// TwinCAT 3 PLC project PLCStudent
// ProgramVersion: 3.1.4026.20
// libraries:
//   Tc2_Standard, * (Beckhoff Automation GmbH)
//   Tc2_System, * (Beckhoff Automation GmbH)
//   Tc2_Utilities, * (Beckhoff Automation GmbH)
//   Tc3_IotBase, * (Beckhoff Automation GmbH)
//   Tc3_JsonXml, * (Beckhoff Automation GmbH)
//   Tc3_Module, * (Beckhoff Automation GmbH)
//   VisuSymbols, 4.5.0.0 (System)
// project tree:
//   / GlobalTextList.TcGTLO, PlcTask.TcTTO, Visualization Manager.TcVMO (not stored)
//   GVLs/ GVL.TcGVL
//   POUs/ FB_HTTP_Get.TcPOU, FB_HTTP_GetSafety.TcPOU, FB_HTTP_Post.TcPOU, FB_OrderAGV.TcPOU, FB_ParseJsonResponse.TcPOU, MAIN.TcPOU, OrderRobot.TcPOU, Process.TcPOU
//   VISUs/ Visualization.TcVIS
// (motion and I/O tree: see PLC project plcsim)
// real-time tasks:
//   TASK PlcTask: cycle T#20ms, priority 20, ADS port 350
// variable links:
//   PLCSim/PLCSim Instance <-> PLCStudent/PLCStudent Instance
//     PlcTask Inputs/GVL.iiGotoPos <-> PlcTask Outputs/GVL.qiGotoPos
//     PlcTask Inputs/GVL.ixPLCStrobe <-> PlcTask Outputs/GVL.qxPLCStrobe
//     PlcTask Outputs/GVL.qiAtPos <-> PlcTask Inputs/GVL.iiAtPos
//     PlcTask Outputs/GVL.qxAGVStrobe <-> PlcTask Inputs/GVL.ixAGVStrobe

CONFIGURATION PLCStudent
    RESOURCE PLC ON TwinCAT3
        TASK PlcTask(INTERVAL := T#20ms, PRIORITY := 20);
        PROGRAM MAIN WITH PlcTask : MAIN;
    END_RESOURCE
END_CONFIGURATION

// ---- GVLs/GVL.TcGVL
{attribute 'qualified_only'}
VAR_GLOBAL
//Input to PLC from process
	ixAGVStrobe		AT %I*:	BOOL;	(* AGV strobe signal *)
	iiAtPos			AT %I*:	INT;	(* Actual position of AGV *)
	
//Output from PLC to process
	qxPLCStrobe		AT %Q*:	BOOL;	(* PLC strobe signal *)
	qiGotoPos		AT %Q*:	INT;	(* Target position for AGV *)
// ADD THESE for R1 route control
    xStart         : BOOL := FALSE;
    iOrder         : INT  := 0;
    xStop          : BOOL := FALSE;
	OrderRobot_0   : OrderRobot;
// R2 data transmission
    sLocation      : STRING := '';
    iBattery       : INT    := 75;
    xSendNow       : BOOL   := FALSE;
END_VAR

// ---- POUs/MAIN.TcPOU
PROGRAM MAIN
VAR
    (* R1: Route state machine *)
    iRouteState     : INT := 0;
    iBattery        : INT := 100;

    (* R2: HTTP POST *)
    fbHttpClientPost : FB_IotHttpClient := (
        sHostName          := '127.0.0.1',
        nHostPort          := 5000,
        bKeepAlive         := TRUE,
        tConnectionTimeout := T#10S
    );
    fbPost      : FB_HTTP_Post;
    bSendPost   : BOOL := FALSE;
    sLocation   : STRING;
   fbFormat : FB_FormatString;
    (* R2: Timestamp *)
    fbTime      : FB_LocalSystemTime := (bEnable := TRUE, dwCycle := 1);
    sTimeStamp  : STRING;

    (* R4: Safety check *)
    fbHttpClientGet : FB_IotHttpClient := (
        sHostName          := '127.0.0.1',
        nHostPort          := 5000,
        bKeepAlive         := TRUE,
        tConnectionTimeout := T#10S
    );
    fbSafetyCheck   : FB_HTTP_GetSafety;
    bSendSafety     : BOOL := FALSE;
    safetyPollTimer : TON;
    sNextLocation   : STRING;
END_VAR

(* R2: 每个周期构建时间戳 *)
fbTime(bEnable := TRUE, dwCycle := 1);
fbFormat(
    sFormat := '%d-%02d-%02d %02d:%02d:%02d', 
    arg1 := F_WORD(fbTime.systemTime.wYear),
    arg2 := F_WORD(fbTime.systemTime.wMonth),
    arg3 := F_WORD(fbTime.systemTime.wDay),
    arg4 := F_WORD(fbTime.systemTime.wHour),
    arg5 := F_WORD(fbTime.systemTime.wMinute),
    arg6 := F_WORD(fbTime.systemTime.wSecond),
    sOut => sTimeStamp
);
CASE iRouteState OF

    (* ────────────────────────────────── *)
    (* 启动阶段                            *)
    (* ────────────────────────────────── *)
    0: (* 启动 — 首先返回原点(Home) *)
        GVL.iOrder  := 1;
        GVL.xStart  := TRUE;
        iRouteState := 10;

    10: (* 等待 AGV 到达原点 *)
        GVL.xStart := FALSE;
        IF GVL.OrderRobot_0.iPhase = 0 THEN
            iRouteState := 12;
        END_IF

    (* ────────────────────────────────── *)
    (* 位置 A                             *)
    (* ────────────────────────────────── *)
    11: (* 前往位置 A *)
        GVL.iOrder  := 2;
        GVL.xStart  := TRUE;
        iRouteState := 20;

    (* ────────────────────────────────── *)
    (* 安全检查 A                         *)
    (* ────────────────────────────────── *)
    12: (* 设置位置，复位发送信号 *)
        sNextLocation := 'A';
        bSendSafety   := FALSE;
        iRouteState   := 13;

    13: (* 发送持续一个周期的脉冲信号 *)
        bSendSafety := TRUE;
        iRouteState := 14;

    14: (* 等待位置 A 的安全检查结果 *)
        bSendSafety := FALSE;
        IF fbSafetyCheck.bDone THEN 
            IF fbSafetyCheck.bIsSafe THEN
                safetyPollTimer(IN := FALSE);
                iRouteState := 11;      (* 安全 → 前往位置 A *)
            ELSE
                (* 不安全 → 等待 2 秒后重试 *)
                safetyPollTimer(IN := TRUE, PT := T#2S);
                IF safetyPollTimer.Q THEN
                    safetyPollTimer(IN := FALSE);
                    iRouteState := 12;  (* 重试 *)
                END_IF
            END_IF
        ELSE
            (* 未收到完成信号 (bDone) → 5 秒后超时 *)
            safetyPollTimer(IN := TRUE, PT := T#5S);
            IF safetyPollTimer.Q THEN
                safetyPollTimer(IN := FALSE);
                iRouteState := 12;      (* 从头重试 *)
            END_IF
        END_IF



    20: (* AGV 已到达位置 A *)
        GVL.xStart := FALSE;
        IF GVL.OrderRobot_0.iPhase = 0 THEN
            sLocation   := 'A';
            iBattery    := iBattery - 5;
            bSendPost   := TRUE;
            iRouteState := 25;
        END_IF

    25: (* 等待位置 A 的 POST 数据上报完成 *)
        bSendPost := FALSE;
        IF NOT fbPost.bBusy THEN
            iRouteState := 26;
        END_IF

    (* ────────────────────────────────── *)
    (* 安全检查 B                         *)
    (* ────────────────────────────────── *)
    26: (* 设置位置，复位发送信号 *)
        sNextLocation := 'B';
        bSendSafety   := FALSE;
        iRouteState   := 27;

    27: (* 发送持续一个周期的脉冲信号 *)
        bSendSafety := TRUE;
        iRouteState := 28;

    28: (* 等待位置 B 的安全检查结果 *)
        bSendSafety := FALSE;
        IF fbSafetyCheck.bDone THEN
            IF fbSafetyCheck.bIsSafe THEN
                safetyPollTimer(IN := FALSE);
                iRouteState := 21;      (* 安全 → 前往位置 B *)
            ELSE
                (* 不安全 → 等待 2 秒后重试 *)
                safetyPollTimer(IN := TRUE, PT := T#2S);
                IF safetyPollTimer.Q THEN
                    safetyPollTimer(IN := FALSE);
                    iRouteState := 26;  (* 重试 *)
                END_IF
            END_IF
        ELSE
            (* 未收到完成信号 (bDone) → 5 秒后超时 *)
            safetyPollTimer(IN := TRUE, PT := T#5S);
            IF safetyPollTimer.Q THEN
                safetyPollTimer(IN := FALSE);
                iRouteState := 26;      (* 从头重试 *)
            END_IF
        END_IF

    (* ────────────────────────────────── *)
    (* 位置 B                             *)
    (* ────────────────────────────────── *)
    21: (* 前往位置 B *)
        GVL.iOrder  := 3;
        GVL.xStart  := TRUE;
        iRouteState := 30;

    30: (* AGV 已到达位置 B *)
        GVL.xStart := FALSE;
        IF GVL.OrderRobot_0.iPhase = 0 THEN
            sLocation   := 'B';
            iBattery    := iBattery - 5;
            bSendPost   := TRUE;
            iRouteState := 35;
        END_IF

    35: (* 等待位置 B 的 POST 数据上报完成 *)
        bSendPost := FALSE;
        IF NOT fbPost.bBusy THEN
            iRouteState := 36;
        END_IF

    (* ────────────────────────────────── *)
    (* 安全检查 C                         *)
    (* ────────────────────────────────── *)
    36: (* 设置位置，复位发送信号 *)
        sNextLocation := 'C';
        bSendSafety   := FALSE;
        iRouteState   := 37;

    37: (* 发送持续一个周期的脉冲信号 *)
        bSendSafety := TRUE;
        iRouteState := 38;

    38: (* 等待位置 C 的安全检查结果 *)
        bSendSafety := FALSE;
        IF fbSafetyCheck.bDone THEN
            IF fbSafetyCheck.bIsSafe THEN
                safetyPollTimer(IN := FALSE);
                iRouteState := 31;      (* 安全 → 前往位置 C *)
            ELSE
                (* 不安全 → 等待 2 秒后重试 *)
                safetyPollTimer(IN := TRUE, PT := T#2S);
                IF safetyPollTimer.Q THEN
                    safetyPollTimer(IN := FALSE);
                    iRouteState := 36;  (* 重试 *)
                END_IF
            END_IF
        ELSE
            (* 未收到完成信号 (bDone) → 5 秒后超时 *)
            safetyPollTimer(IN := TRUE, PT := T#5S);
            IF safetyPollTimer.Q THEN
                safetyPollTimer(IN := FALSE);
                iRouteState := 36;      (* 从头重试 *)
            END_IF
        END_IF

    (* ────────────────────────────────── *)
    (* 位置 C                             *)
    (* ────────────────────────────────── *)
    31: (* 前往位置 C *)
        GVL.iOrder  := 4;
        GVL.xStart  := TRUE;
        iRouteState := 40;

    40: (* AGV 已到达位置 C *)
        GVL.xStart := FALSE;
        IF GVL.OrderRobot_0.iPhase = 0 THEN
            sLocation   := 'C';
            iBattery    := iBattery - 5;
            bSendPost   := TRUE;
            iRouteState := 45;
        END_IF

    45: (* 等待位置 C 的 POST 数据上报完成 *)
        bSendPost := FALSE;
        IF NOT fbPost.bBusy THEN
            iRouteState := 46;
        END_IF

    (* ────────────────────────────────── *)
    (* 安全检查 D                         *)
    (* ────────────────────────────────── *)
    46: (* 设置位置，复位发送信号 *)
        sNextLocation := 'D';
        bSendSafety   := FALSE;
        iRouteState   := 47;

    47: (* 发送持续一个周期的脉冲信号 *)
        bSendSafety := TRUE;
        iRouteState := 48;

    48: (* 等待位置 D 的安全检查结果 *)
        bSendSafety := FALSE;
        IF fbSafetyCheck.bDone THEN
            IF fbSafetyCheck.bIsSafe THEN
                safetyPollTimer(IN := FALSE);
                iRouteState := 41;      (* 安全 → 前往位置 D *)
            ELSE
                (* 不安全 → 等待 2 秒后重试 *)
                safetyPollTimer(IN := TRUE, PT := T#2S);
                IF safetyPollTimer.Q THEN
                    safetyPollTimer(IN := FALSE);
                    iRouteState := 46;  (* 重试 *)
                END_IF
            END_IF
        ELSE
            (* 未收到完成信号 (bDone) → 5 秒后超时 *)
            safetyPollTimer(IN := TRUE, PT := T#5S);
            IF safetyPollTimer.Q THEN
                safetyPollTimer(IN := FALSE);
                iRouteState := 46;      (* 从头重试 *)
            END_IF
        END_IF

    (* ────────────────────────────────── *)
    (* 位置 D                             *)
    (* ────────────────────────────────── *)
    41: (* 前往位置 D *)
        GVL.iOrder  := 5;
        GVL.xStart  := TRUE;
        iRouteState := 50;

    50: (* AGV 已到达位置 D *)
        GVL.xStart := FALSE;
        IF GVL.OrderRobot_0.iPhase = 0 THEN
            sLocation   := 'D';
            iBattery    := iBattery - 5;
            bSendPost   := TRUE;
            iRouteState := 55;
        END_IF

    55: (* 等待位置 D 的 POST 数据上报完成 *)
        bSendPost := FALSE;
        IF NOT fbPost.bBusy THEN
            iRouteState := 51;
        END_IF

    (* ────────────────────────────────── *)
    (* 返回原点                            *)
    (* ────────────────────────────────── *)
    51: (* 返回原点(Home) *)
        GVL.iOrder  := 1;
        GVL.xStart  := TRUE;
        iRouteState := 60;

    60: (* AGV 已到达原点 — 进行充电 *)
        GVL.xStart := FALSE;
        IF GVL.OrderRobot_0.iPhase = 0 THEN
            sLocation   := 'Home';
            iBattery    := 100;
            bSendPost   := TRUE;
            iRouteState := 65;
        END_IF

    65: (* 等待原点的 POST 数据上报完成 — 再次进入循环 *)
        bSendPost := FALSE;
        IF NOT fbPost.bBusy THEN
            iRouteState := 12;  (* 从位置 A 的安全检查重新开始循环 *)
        END_IF

END_CASE

(* ────────────────────────────────────── *)
(* 始终在每个周期执行                      *)
(* ────────────────────────────────────── *)
fbHttpClientPost.Execute();
fbHttpClientGet.Execute();

fbPost(
    bSend    := bSendPost,
    position := sLocation,
    dateTime := sTimeStamp,
    battery  := iBattery,
    fbClient := fbHttpClientPost
);

fbSafetyCheck(
    bSend     := bSendSafety,
    sLocation := sNextLocation,
    fbClient  := fbHttpClientGet
);

Process();

END_PROGRAM

// ---- POUs/FB_HTTP_Post.TcPOU
FUNCTION_BLOCK FB_HTTP_Post
VAR_INPUT
    bSend           : BOOL;             //Trigger send message
    position        : STRING;           //Location A, B, C, D, Home
    dateTime        : STRING;           //Timestamp
    battery         : INT;              //Battery level
END_VAR
VAR_IN_OUT
    fbClient        : FB_IotHttpClient;
END_VAR
VAR_OUTPUT
    bBusy           : BOOL;
    bError          : BOOL;
    nResCount       : UDINT;
    nOutputStatusCode : UINT;
    sOutputMessage  : STRING(511);
END_VAR
VAR
    fbRequest       : FB_IotHttpRequest;
    fbJson          : FB_JsonDomParser;
    fbPayload       : FB_JsonSaxWriter;
    fbHeader        : FB_IotHttpHeaderFieldMap;
    RisingEdge      : R_TRIG;
    nState          : UDINT;
    bGetContentResult : BOOL;
    sContent        : STRING(511);
    nReqCount       : UDINT;
    nErrCount       : UDINT;
    LoggMessage     : STRING;
	sBattery : STRING;
END_VAR

RisingEdge(CLK:= bSend);
CASE nState OF
0:
    IF RisingEdge.Q THEN
        sContent := DELETE(STR:=sContent, LEN:=511, POS:=1);
        fbPayload.ResetDocument();
        fbPayload.StartObject();
        fbHeader.AddField('Content-Type', 'application/json', FALSE);

        (* Position *)
        fbPayload.AddKey('Position');
        fbPayload.AddString(position);

        (* TimeStamp — no colon! *)
        fbPayload.AddKey('TimeStamp');
        fbPayload.AddString(dateTime);

        (* Battery — NEW *)
        sBattery := INT_TO_STRING(battery);
        fbPayload.AddKey('Battery');
        fbPayload.AddString(sBattery);

        fbPayload.EndObject();
        sContent := fbPayload.GetDocument();

        IF fbRequest.SendRequest(
            sUri         := '/post_data',
            fbClient     := fbClient,
            eRequestType := ETcIotHttpRequestType.HTTP_POST,
            pContent     := ADR(sContent),
            nContentSize := LEN2(ADR(sContent)),
            fbHeader) THEN

            nState   := 1;
            IF nReqCount > 10 THEN
                nReqCount := 0;
            END_IF
            nReqCount := nReqCount + 1;
            bBusy     := TRUE;
            bError    := FALSE;
        END_IF
    END_IF

1:
    IF NOT fbRequest.bBusy THEN
        bError            := TRUE;
        nOutputStatusCode := fbRequest.nStatusCode;

        IF NOT fbRequest.bError THEN
            bGetContentResult := fbRequest.GetContent(
                pContent           := ADR(sContent),
                nContentSize       := SIZEOF(sContent),
                bSetNullTermination := TRUE);

            sOutputMessage := sContent;

            IF fbRequest.nStatusCode >= 200 AND fbRequest.nStatusCode < 300 THEN
                bError    := FALSE;
                nResCount := nResCount + 1;
                bBusy     := FALSE;
            END_IF
        END_IF

        nState := 0;
        IF bError THEN
            nErrCount := nErrCount + 1;
        END_IF
    END_IF
END_CASE

END_FUNCTION_BLOCK

// ---- POUs/FB_HTTP_GetSafety.TcPOU
FUNCTION_BLOCK FB_HTTP_GetSafety
VAR_INPUT
    bSend           : BOOL;
    sLocation       : STRING;    (* Pass 'A', 'B', 'C' or 'D' *)
END_VAR
VAR_IN_OUT
    fbClient        : FB_IotHttpClient;
END_VAR
VAR_OUTPUT
    bBusy           : BOOL;
    bError          : BOOL;
    bDone           : BOOL;
    nOutputStatusCode : UINT;
    bIsSafe         : BOOL;      (* TRUE = safe, FALSE = unsafe *)
END_VAR
VAR
    fbRequest       : FB_IotHttpRequest;
    fbJson          : FB_JsonDomParser;
    nState          : UDINT;
    RisingEdge      : R_TRIG;
    jsonDoc         : SJsonValue;
    jsonVal         : SJsonValue;
    sResultValue    : STRING;
    sFullUri        : STRING;
    LoggMessage     : STRING;
END_VAR

RisingEdge(CLK := bSend);  // 调用上升沿检测功能块，把输入CLK绑定到bSend信号，用于检测从FALSE→TRUE的瞬间

CASE nState OF   // 状态机，根据当前状态nState执行不同逻辑

0:  // 状态0：空闲/准备发送请求状态
    bDone := FALSE;  // 标记当前任务尚未完成（每次进入初始状态都清零完成标志）
    
    IF RisingEdge.Q THEN  // 如果检测到bSend的上升沿（触发一次请求）
        
        (* Only path, not full URL *)  // 注释说明这里只拼接路径，不是完整URL
        sFullUri := CONCAT('/get_safety/', sLocation);  // 拼接请求路径，例如 /get_safety/A1

        IF fbRequest.SendRequest(  // 调用HTTP请求发送函数
            sUri         := sFullUri,  // 请求的URI路径
            fbClient     := fbClient,  // HTTP客户端实例
            eRequestType := ETcIotHttpRequestType.HTTP_GET,  // 请求类型：GET
            0, 0, 0)  // 额外参数（未使用，占位）
        THEN  // 如果请求成功发起（注意：只是“发出去”，不是“收到响应”）
            
            nState := 1;  // 切换到状态1（等待响应）
            bBusy  := TRUE;  // 标记系统正在忙（请求处理中）
            bError := FALSE;  // 清除错误标志
            bDone  := FALSE;  // 再次确认未完成（其实这里有点重复）

            ADSLOGSTR(  // TwinCAT日志输出函数
                msgCtrlMask := ADSLOG_MSGTYPE_HINT,  // 日志类型：提示信息
                msgFmtStr   := 'SafetyCheck: Sending request for location %s',  // 日志格式字符串
                strArg      := sLocation  // 替换%s的参数（位置名）
            );
        END_IF
    END_IF

1:  // 状态1：等待HTTP响应完成
    IF NOT fbRequest.bBusy THEN  // 如果请求已经处理完成（不再忙）
        
        nOutputStatusCode := fbRequest.nStatusCode;  // 保存HTTP返回状态码（例如200、404等）

        IF NOT fbRequest.bError AND  // 如果请求过程中没有错误
           fbRequest.nStatusCode >= 200 AND  // 且HTTP状态码在200以上
           fbRequest.nStatusCode < 300  // 且小于300（表示成功响应）
        THEN
            
            jsonDoc := fbRequest.GetJsonDomContent(fbJson);  // 解析HTTP响应内容为JSON DOM结构

            IF jsonDoc <> 0 THEN  // 如果JSON解析成功（非空指针）
                
                (* server.py returns {"safe": "true"} or {"safe": "false"} *)  // 服务端返回格式说明
                
                jsonVal      := fbJson.FindMember(jsonDoc, 'safe');  // 在JSON中查找字段 "safe"
                sResultValue := fbJson.GetString(jsonVal);  // 获取该字段的字符串值（"true" 或 "false"）

                IF sResultValue = 'true' THEN  // 如果返回值是字符串"true"
                    bIsSafe := TRUE;  // 标记为安全
                ELSE  // 否则（包括"false"或异常情况）
                    bIsSafe := FALSE;  // 标记为不安全
                END_IF

                LoggMessage := sResultValue;  // 保存结果字符串用于日志输出
                
                ADSLOGSTR(  // 输出日志
                    msgCtrlMask := ADSLOG_MSGTYPE_HINT,  // 提示类型日志
                    msgFmtStr   := 'SafetyCheck result: %s',  // 日志格式
                    strArg      := LoggMessage  // 输出实际返回值
                );
            ELSE  // 如果JSON解析失败
                
                bIsSafe := FALSE;  // 默认认为不安全（保守处理）
                bError  := TRUE;  // 标记发生错误
            END_IF
        
        ELSE  // 如果请求失败（HTTP错误或通信错误）
            
            bIsSafe := FALSE;  // 默认不安全
            bError  := TRUE;  // 标记错误
        END_IF

        bDone  := TRUE;  // 标记任务完成（无论成功失败都会置TRUE）
        bBusy  := FALSE;  // 清除忙状态
        nState := 0;  // 回到初始状态，等待下一次触发
    END_IF

END_CASE  // 状态机结束

END_FUNCTION_BLOCK

// ---- POUs/Process.TcPOU
PROGRAM Process
VAR
	OrderRobot_0: OrderRobot;
	xStart: BOOL;
	iOrder: INT;
	xStop: BOOL;
END_VAR

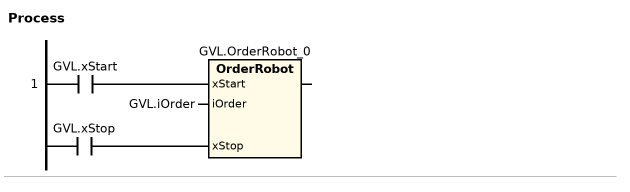
// NETWORK 1
GVL.OrderRobot_0(xStart := GVL.xStart, iOrder := GVL.iOrder, xStop := GVL.xStop); // OrderRobot

END_PROGRAM

// ---- POUs/OrderRobot.TcPOU
FUNCTION_BLOCK OrderRobot
VAR_INPUT
	xStart: BOOL;
	iOrder: INT;
	xStop: BOOL;
END_VAR
VAR_OUTPUT
END_VAR
VAR
	iPhase: INT:=0; //0: Wait signal
END_VAR

CASE iPhase OF
	0: // Wait signal
		IF xStart AND (iOrder<>0) THEN
			iPhase:=1;
		END_IF
	1: // Set Order, here you can add more checking of the numbers are legal or not
		GVL.qiGotoPos:=iOrder;
		iPhase:=2;
	2: // Set strobe
		GVL.qxPLCStrobe:=TRUE;
		iPhase:=3;
	3: // Wait for input strobe
		IF gvl.ixAGVStrobe THEN
			gvl.qiGotoPos:=0;
			gvl.qxPLCStrobe:=FALSE;
			iPhase:=4;
		END_IF
	4: // wait for order finish or stop
		IF xStop THEN
			iPhase:=5;
		ELSIF gvl.iiAtPos<>0 THEN
			iPhase:=6;
		END_IF
	5: // Try to stop
		gvl.qiGotoPos:=6;
		iPhase:=12;
	6: //Wait strobe
		IF gvl.ixAGVStrobe THEN
			iPhase:=7;
		END_IF
	7: // Set strobe
		gvl.qxPLCStrobe:=TRUE;
		iPhase:=8;
	8: // wait for reset
		IF gvl.iiAtPos=0 AND (NOT gvl.ixAGVStrobe) THEN
			gvl.qxPLCStrobe:=FALSE;
			iphase:=0;
		END_IF
	12: // Set strobe
		GVL.qxPLCStrobe:=TRUE;
		iPhase:=13;
	13: // Wait for input strobe
		IF gvl.ixAGVStrobe THEN
			gvl.qiGotoPos:=0;
			gvl.qxPLCStrobe:=FALSE;
			iPhase:=14;
		END_IF
	14: // wait for order finish or stop
		IF gvl.iiAtPos=6 THEN
			iPhase:=16;
		END_IF
	16: //Wait strobe
		IF gvl.ixAGVStrobe THEN
			iPhase:=17;
		END_IF
	17: // Set strobe
		gvl.qxPLCStrobe:=TRUE;
		iPhase:=18;
	18: // wait for reset
		IF gvl.iiAtPos=0 AND (NOT gvl.ixAGVStrobe) THEN
			gvl.qxPLCStrobe:=FALSE;
			iphase:=19;
		END_IF
	19: // Go home
		GVL.qiGotoPos:=1;
		iPhase:=2;
END_CASE

END_FUNCTION_BLOCK

// ---- POUs/FB_HTTP_Get.TcPOU
FUNCTION_BLOCK FB_HTTP_Get
VAR_INPUT
	bSend				: BOOL;
END_VAR
VAR_IN_OUT
	fbClient			: FB_IotHttpClient;
END_VAR	
VAR_OUTPUT
	bBusy				: BOOL;
	bError				: BOOL;
	nOutputStatusCode   : UINT;
	sOutputMessage      : STRING(511);
END_VAR
VAR	
	fbRequest			: FB_IotHttpRequest;
	fbJson				: FB_JsonDomParser;
	jsonMember       : SJsonValue;
	fbHeader: FB_IotHttpHeaderFieldMap;
	nState				: UDINT;
	RisingEdge			: R_TRIG;
	
	bGetContentResult	: BOOL;
	sContent			: STRING(2000);
	
	bGetJsonResult		: BOOL;
	jsonDoc				: SJsonValue;
	jsonVal				: SJsonValue;
	sResultValue		: STRING;
	
	
	nReqCount			: UDINT;
	nResCount			: UDINT;
	nValidResCount		: UDINT;
	nErrCount			: UDINT;	
	LoggMessage			:STRING;		(*Debugger varible*)
	jsonString: STRING(255);
	uValue: LREAL;
	sUri: STRING;
END_VAR

RisingEdge(CLK:= bSend);
CASE nState OF
0:		
	IF RisingEdge.Q THEN
		IF fbRequest.SendRequest(sUri:='/get_variable/example_var2', fbClient:= fbClient, eRequestType:= ETcIotHttpRequestType.HTTP_GET, 0, 0, 0) THEN				
			nState:= 1;
			nReqCount:= nReqCount+1;
			bBusy:= TRUE;
			bError:= FALSE;
			
			LoggMessage:='';
			ADSLOGSTR(
				msgCtrlMask := ADSLOG_MSGTYPE_HINT, 
				msgFmtStr   := 'Get 0:1', 
				strArg      := LoggMessage
			);
		END_IF					
	END_IF
1:
	IF NOT fbRequest.bBusy THEN
		bError:= TRUE;
		
		// 1. HTTP state to var
		nOutputStatusCode := fbRequest.nStatusCode;
		
		ADSLOGSTR(
			msgCtrlMask := ADSLOG_MSGTYPE_HINT, 
			msgFmtStr   := 'Get 1:1', 
			strArg      := ''
		);
		
		IF NOT fbRequest.bError THEN	
			ADSLOGSTR(
				msgCtrlMask := ADSLOG_MSGTYPE_HINT, 
				msgFmtStr   := 'Get 1:2 %s', 
				strArg      := sContent
			);			 
			LoggMessage:=INT_TO_STRING(len(sContent));
			ADSLOGSTR(
				msgCtrlMask := ADSLOG_MSGTYPE_HINT, 
				msgFmtStr   := 'lenght of string is %s', 
				strArg      := LoggMessage
			);	
			
			//sContent:=DELETE(STR:=sContent , LEN:=511 , POS:=1 );		
			//bGetContentResult:= fbRequest.GetContent(pContent:= ADR(sContent), nContentSize:= SIZEOF(sContent), bSetNullTermination:= TRUE);	
			
			// 2. String to var
			//sOutputMessage := sContent;
			
			IF fbRequest.nStatusCode >= 200 AND fbRequest.nStatusCode < 300 THEN
				bGetJsonResult:= FALSE;
				jsonDoc:= fbRequest.GetJsonDomContent(fbJson);	
				sOutputMessage :=fbJson.GetString(jsonDoc);		
				IF jsonDoc <> 0 THEN		
					jsonVal := fbJson.FindMember(jsonDoc, 'example_var2');					
					sResultValue := fbJson.GetString(jsonVal);
					uValue := STRING_TO_LREAL(sResultValue);
					//jsonVal := fbJson.FindMember(jsonDoc, 'example_var1');					
					//sResultValue := fbJson.GetString(jsonVal);

					ADSLOGSTR((*Debugger*)
						msgCtrlMask := ADSLOG_MSGTYPE_HINT, 
						msgFmtStr   := 'jsonDoc get message is: %s', 
						strArg      := sResultValue
					);
					nValidResCount:= nValidResCount+1;
					bError:= FALSE;
				END_IF
				nResCount:= nResCount+1;					
			END_IF				
		END_IF
		
		nState:= 0;
		bBusy:= FALSE;
		IF bError THEN
			nErrCount:= nErrCount+1;
		END_IF		
	END_IF  	
END_CASE

END_FUNCTION_BLOCK

// ---- POUs/FB_OrderAGV.TcPOU
FUNCTION_BLOCK FB_OrderAGV
VAR_INPUT
	xStart: BOOL;
	iOrder: INT;
END_VAR
VAR_OUTPUT
END_VAR
VAR
	iState: INT :=0; // 0 is init state
END_VAR

CASE iState OF
	0: // init
		IF xStart AND (iOrder<>0) THEN
			iState:=1;
		END_IF
	1: // Send order
		gvl.qiGotoPos:=iOrder;
		iState:=2;
	2: //Set strobe
		gvl.qxPLCStrobe:=TRUE;
		IF gvl.ixAGVStrobe THEN
			iState:=3;
		END_IF
	3: //Order recieved
		gvl.qiGotoPos:=0;
		gvl.qxPLCStrobe:=FALSE;
		IF gvl.iiAtPos<>0 THEN
			iState:=4;
		END_IF
	4: //Wait for strobe
		IF gvl.ixAGVStrobe THEN
			iState:=5;
		END_IF
	5: //AGV moved
		gvl.qxPLCStrobe:=TRUE;
		IF (NOT gvl.ixAGVStrobe) AND gvl.iiAtPos=0 THEN
			iState:=6;
		END_IF
	6: //Answer ready
		iState:=0;
END_CASE

END_FUNCTION_BLOCK

// ---- POUs/FB_ParseJsonResponse.TcPOU
FUNCTION_BLOCK FB_ParseJsonResponse
VAR_INPUT
	bExecute    : BOOL; 
    sJsonString : STRING(511); 
           
END_VAR

VAR_OUTPUT
	bDone       : BOOL;   
    sMessage    : STRING(255); // Extracted "message"
    fPosition   : LREAL;       // Converted "Position"
    sTimeStamp  : STRING(255); // Extracted "TimeStamp:" 
    bError      : BOOL;        
END_VAR

VAR
    fbJsonParser     : FB_JsonDomParser;
    jsonDoc          : SJsonValue;
    jsonMember       : SJsonValue;
    jsonNodeYourData : SJsonValue; // Node to hold the "your_data" object
    rtExecute        : R_TRIG;
    
    sTempPosition    : STRING(255); // Temporary string for conversion
END_VAR

rtExecute(CLK := bExecute);  // 上升沿触发检测功能块，把输入CLK绑定到bExecute，用于检测执行信号的上升沿

IF rtExecute.Q THEN  // 如果检测到bExecute从FALSE→TRUE的上升沿（只触发一次）
    bDone  := FALSE;  // 清除完成标志，表示当前解析任务尚未完成
    bError := FALSE;  // 清除错误标志，表示开始时默认没有错误
    
    // Parse the incoming string (TwinCAT handles the $N newline characters automatically)
    jsonDoc := fbJsonParser.ParseDocument(sJsonString);  // 解析输入的JSON字符串sJsonString，生成JSON文档结构（DOM）
    
    IF jsonDoc <> 0 THEN  // 如果解析成功（返回的JSON文档句柄不=0）
        
        // 1. Extract the root-level "message"
        jsonMember := fbJsonParser.FindMember(jsonDoc, 'message');  // 在JSON根节点中查找字段 "message"
        IF jsonMember <> 0 THEN  // 如果成功找到该字段 
            sMessage := fbJsonParser.GetString(jsonMember); // 获取该字段的字符串值并赋给sMessage
        END_IF
        
        // 2. Locate the nested "your_data" object
        jsonNodeYourData := fbJsonParser.FindMember(jsonDoc, 'your_data'); // 在JSON根节点中查找嵌套对象 "your_data"
        
        IF jsonNodeYourData <> 0 THEN
            
            // 3. Extract "Position" from INSIDE "your_data"
            jsonMember := fbJsonParser.FindMember(jsonNodeYourData, 'Position'); // 在内部查找字段 "Position"
            IF jsonMember <> 0 THEN // 如果找到Position字段
                sTempPosition := fbJsonParser.GetString(jsonMember);  // 获取Position的字符串值（例如 "10"）
                fPosition     := STRING_TO_LREAL(sTempPosition); // Convert string "10" to LREAL 10.0
            END_IF
            
            // 4. Extract "TimeStamp:" from INSIDE "your_data" (Note the included colon)
            jsonMember := fbJsonParser.FindMember(jsonNodeYourData, 'TimeStamp'); // 在查找字段 "TimeStamp:"（注意字段名包含冒号）
            IF jsonMember <> 0 THEN
                sTimeStamp := fbJsonParser.GetString(jsonMember); // 获取时间戳字符串值并赋给sTimeStamp
            END_IF
            
        END_IF
        
        bDone := TRUE; // JSON解析和数据提取完成，设置完成标志为TRUE
    ELSE               // 如果JSON解析失败（jsonDoc为0）
        bError := TRUE;   // 设置错误标志，表示解析过程中出现问题
    END_IF
END_IF

END_FUNCTION_BLOCK

// ---- VISUs/Visualization.TcVIS
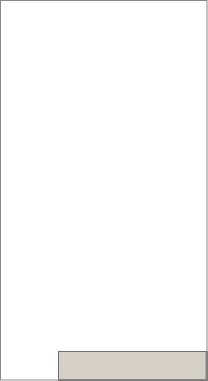
VISUALIZATION Visualization  // 208x381
    Button (58,351 150x30)
        tap Process.xStop
END_VISUALIZATION
